// TIA Portal project "Grundkurs Aufgabe 10 NEU" (V15.1)
// Vorlageprojekt für das Buch mit Zielsystem S7-1200

(* hardware
DEVICE "S7-1200-Station_1"  S7-1200 Station
   slot 0: "Baugruppenträger_0"  Rack  V1.0
   slot 1: "SPS"  CPU 1212C AC/DC/Rly  6ES7 212-1BE40-0XB0  V4.2
*)

// ===== PLC "SPS"  CPU 1212C AC/DC/Rly =====

VAR_GLOBAL   // PLC tag table "Eingänge und Ausgänge"
   "Sensor_Bauteil_induktiv" AT %E0.0 : Bool;   // Induktiver Sensor für Werkstofferkennung (Schließer)
   "Sensor_Bauteil_kapazitiv" AT %E0.1 : Bool;   // Kapazitiver Sensor für Werkstofferkennung (Schließer)
   "Endlage_Ausschieber_vorne" AT %E0.2 : Bool;   // Ausschieber hat vorderer Endlage erreicht (Schließer)
   "Endlage_Ausschieber_hinten" AT %E0.3 : Bool;   // Ausschieber hat hintere Endlage erreicht (Schließer)
   "Lichttaster_Auslauf_links" AT %E0.4 : Bool;   // Lichttaster auf Förderband Auslauf links (Schließer)
   "Lichttaster_Auslauf_rechts" AT %E0.5 : Bool;   // Lichttaster auf Förderband Auslauf rechts (Schließer)
   "Motor_Foerderband_Einlauf" AT %A0.0 : Bool;   // Motor Förderband Einlauf vorwärts fahren
   "Motor_Foerderband_Auslauf_links" AT %A0.1 : Bool;   // Motor Förderband Auslauf links vorwärts fahren
   "Motor_Foerderband_Auslauf_rechts" AT %A0.2 : Bool;   // Motor Förderband Auslauf rechts vorwärts fahren
   "Ausschieber_vor" AT %A0.3 : Bool;   // Ausschieber nach vorne fahren (1-Signal = ausfahren / 0-Signal = einfahren)
END_VAR

VAR_GLOBAL   // PLC tag table "Merker"
   "Foerderbaender_Einlauf_Auslauf_vor" AT %M1.0 : Bool;   // Förderbänder Einlauf und Auslauf rechts vorwärts fahren
   "Bauteil_Kunststoff_erkannt" AT %M1.1 : Bool;   // Kunststoffbauteil wurde erkannt
   "Bauteil_Metall_erkannt" AT %M1.2 : Bool;   // Metallbauteil wurde erkannt
   "Bauteil_verschieben" AT %M1.3 : Bool;   // Bauteil auf anderes Förderband verschieben
   "Foerderband_Auslauf_links_vor" AT %M1.4 : Bool;   // Förderband Auslauf links vorwärts fahren
   "Foerderband_Auslauf_rechts_vor" AT %M1.5 : Bool;   // Förderband Auslauf rechts vorwärts fahren
   "Hilfsmerker_FN1" AT %M100.0 : Bool;   // Hilfsmerker für negative Flanke
   "Hilfsmerker_FN2" AT %M100.1 : Bool;   // Hilfsmerker für negative Flanke
   "Hilfsmerker_FN3" AT %M100.2 : Bool;   // Hilfsmerker für negative Flanke
   "Hilfsmerker_FN4" AT %M100.3 : Bool;   // Hilfsmerker für negative Flanke
END_VAR

FUNCTION "Kopplung_FactoryIO_mit_PLCSIM" : Void   // FC9000, SCL
{ S7_Optimized_Access := 'TRUE' }
VERSION : 0.1
   VAR_TEMP
      rdTimeReturn : Int;
      outputTime : DTL;
      SyncVal : Byte;
      forVal : Int;
      forVal_2 : Int;
      Value : Byte;
   END_VAR
   VAR CONSTANT
      CompVal : Byte := 16#34;
      Value_01 : Byte := 16#11;
      Value_01_DW : DWord := 16#A165_D992;
      Value_02_DW : DWord := 16#58BE_4401;
   END_VAR
BEGIN

   #Value:=PEEK(area := 16#82,
        dbNumber := 0,
        byteOffset := 511);
   #Value := #Value + 1;

   POKE(area := 16#82,
        dbNumber := 0,
        byteOffset := 511,
        value := #Value);

   POKE(area:=16#81,
        dbNumber:=0,
        byteOffset:=1016,
        value:=#Value_01_DW);
   POKE(area := 16#81,
        dbNumber := 0,
        byteOffset := 1020,
        value := #Value_02_DW);

   POKE(area := 16#81,
        dbNumber := 0,
        byteOffset := 511,
        value := B#16#00);

   FOR #forVal := 0 TO 120 DO
       FOR #forVal_2:=0 TO 10 DO
           #rdTimeReturn:=RD_SYS_T(#outputTime);
           #rdTimeReturn := WR_SYS_T(#outputTime);
           #rdTimeReturn := RD_SYS_T(#outputTime);
           #rdTimeReturn := WR_SYS_T(#outputTime);
       END_FOR;
       #SyncVal:= PEEK(area := 16#81,
                      dbNumber := 0,
                      byteOffset := 511);
       IF #SyncVal = #CompVal THEN
          GOTO M_1;
       END_IF;
   END_FOR;
   RETURN;

   M_1:
   POKE(area := 16#81,
        dbNumber := 0,
        byteOffset := 511,
        value := B#16#0);
END_FUNCTION

ORGANIZATION_BLOCK "Main"   // OB1, FBD, ProgramCycle
TITLE = "Main Program Sweep (Cycle)"
{ S7_Optimized_Access := 'TRUE' }
VERSION : 0.1
   VAR_INPUT
      Initial_Call : Bool;   // Initial call of this OB
      Remanence : Bool;   // =True, if remanent data are available
   END_VAR
   VAR_TEMP   // added for the SCL form of the ladder/FBD networks
      _w1 : Bool;
   END_VAR
BEGIN

REGION Network 1: Konnektierungsbaustein für PLC-Lab / Bausteinaufruf FC9000 (Für Aufgabe nicht relevant)
   // Im Netzwerk 1 wird der Konnektierungsbaustein für PLC-Lab aufgerufen.
   // Dieser Aufruf darf nicht entfernt werden!
   // Der Baustein FC9000 organisiert den Datentransfer zwischen PLCSIM und FactoryIO.
   // Der Baustein kann als Beispielprojekt von der FactoryIO-Homepage heruntergeladen werden.
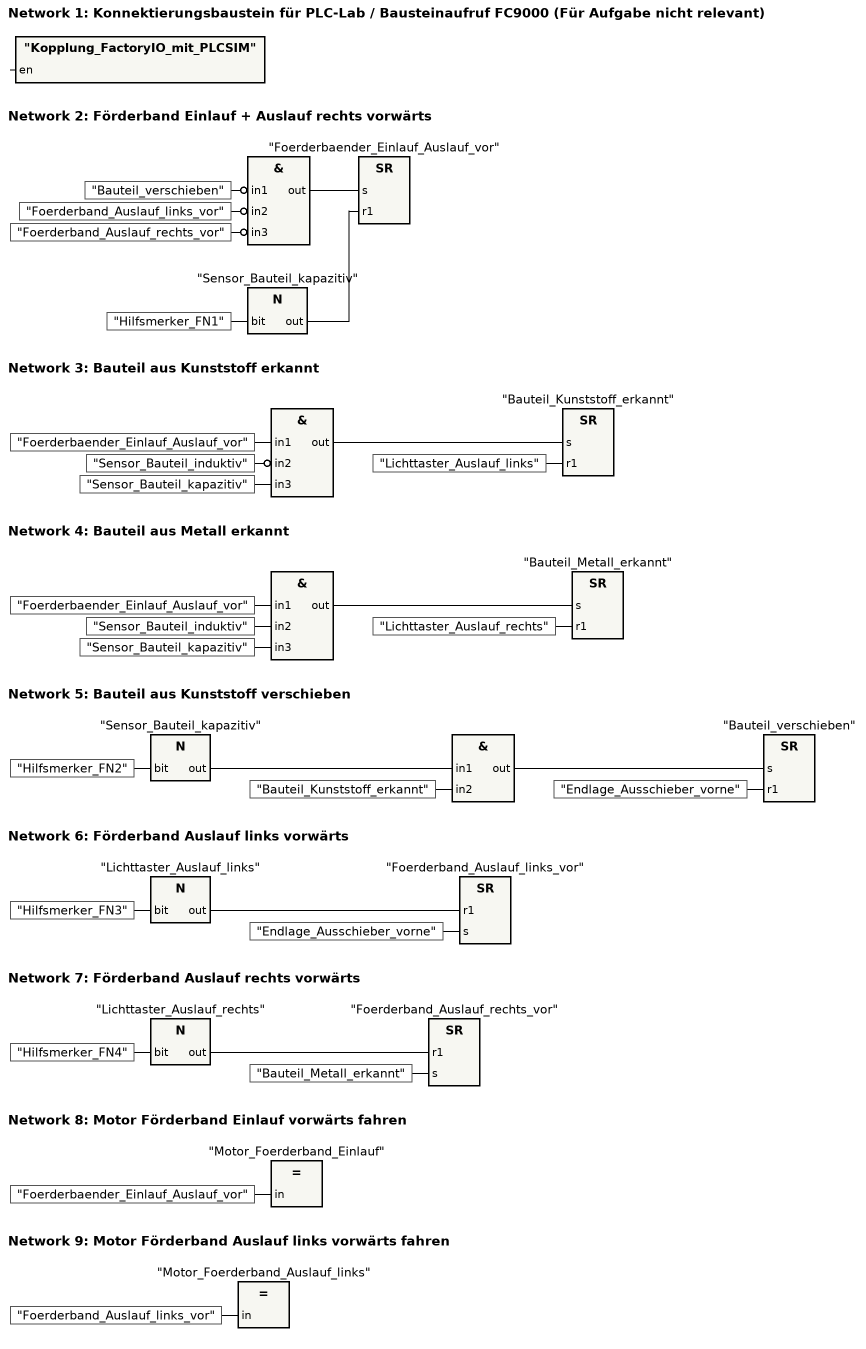
   "Kopplung_FactoryIO_mit_PLCSIM"();
END_REGION

REGION Network 2: Förderband Einlauf + Auslauf rechts vorwärts
   #_w1 := NOT "Sensor_Bauteil_kapazitiv" AND "Hilfsmerker_FN1";   // falling edge of "Sensor_Bauteil_kapazitiv"
   "Hilfsmerker_FN1" := "Sensor_Bauteil_kapazitiv";
   IF NOT "Bauteil_verschieben" AND NOT "Foerderband_Auslauf_links_vor" AND NOT "Foerderband_Auslauf_rechts_vor" THEN
       "Foerderbaender_Einlauf_Auslauf_vor" := TRUE;   // SR flip-flop
   END_IF;
   IF #_w1 THEN "Foerderbaender_Einlauf_Auslauf_vor" := FALSE; END_IF;
END_REGION

REGION Network 3: Bauteil aus Kunststoff erkannt
   IF "Foerderbaender_Einlauf_Auslauf_vor" AND NOT "Sensor_Bauteil_induktiv" AND "Sensor_Bauteil_kapazitiv" THEN
       "Bauteil_Kunststoff_erkannt" := TRUE;   // SR flip-flop
   END_IF;
   IF "Lichttaster_Auslauf_links" THEN "Bauteil_Kunststoff_erkannt" := FALSE; END_IF;
END_REGION

REGION Network 4: Bauteil aus Metall erkannt
   IF "Foerderbaender_Einlauf_Auslauf_vor" AND "Sensor_Bauteil_induktiv" AND "Sensor_Bauteil_kapazitiv" THEN
       "Bauteil_Metall_erkannt" := TRUE;   // SR flip-flop
   END_IF;
   IF "Lichttaster_Auslauf_rechts" THEN "Bauteil_Metall_erkannt" := FALSE; END_IF;
END_REGION

REGION Network 5: Bauteil aus Kunststoff verschieben
   #_w1 := NOT "Sensor_Bauteil_kapazitiv" AND "Hilfsmerker_FN2";   // falling edge of "Sensor_Bauteil_kapazitiv"
   "Hilfsmerker_FN2" := "Sensor_Bauteil_kapazitiv";
   IF #_w1 AND "Bauteil_Kunststoff_erkannt" THEN
       "Bauteil_verschieben" := TRUE;   // SR flip-flop
   END_IF;
   IF "Endlage_Ausschieber_vorne" THEN "Bauteil_verschieben" := FALSE; END_IF;
END_REGION

REGION Network 6: Förderband Auslauf links vorwärts
   #_w1 := NOT "Lichttaster_Auslauf_links" AND "Hilfsmerker_FN3";   // falling edge of "Lichttaster_Auslauf_links"
   "Hilfsmerker_FN3" := "Lichttaster_Auslauf_links";
   IF "Endlage_Ausschieber_vorne" THEN
       "Foerderband_Auslauf_links_vor" := TRUE;   // SR flip-flop
   END_IF;
   IF #_w1 THEN "Foerderband_Auslauf_links_vor" := FALSE; END_IF;
END_REGION

REGION Network 7: Förderband Auslauf rechts vorwärts
   #_w1 := NOT "Lichttaster_Auslauf_rechts" AND "Hilfsmerker_FN4";   // falling edge of "Lichttaster_Auslauf_rechts"
   "Hilfsmerker_FN4" := "Lichttaster_Auslauf_rechts";
   IF "Bauteil_Metall_erkannt" THEN
       "Foerderband_Auslauf_rechts_vor" := TRUE;   // SR flip-flop
   END_IF;
   IF #_w1 THEN "Foerderband_Auslauf_rechts_vor" := FALSE; END_IF;
END_REGION

REGION Network 8: Motor Förderband Einlauf vorwärts fahren
   "Motor_Foerderband_Einlauf" := "Foerderbaender_Einlauf_Auslauf_vor";
END_REGION

REGION Network 9: Motor Förderband Auslauf links vorwärts fahren
   "Motor_Foerderband_Auslauf_links" := "Foerderband_Auslauf_links_vor";
END_REGION

REGION Network 10: Motor Förderband Auslauf rechts vorwärts fahren
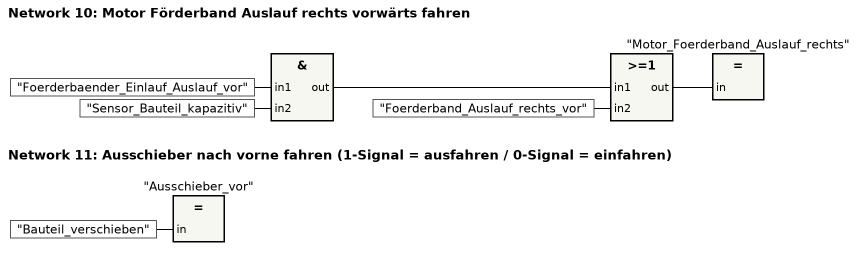
   "Motor_Foerderband_Auslauf_rechts" := ("Foerderbaender_Einlauf_Auslauf_vor" AND "Sensor_Bauteil_kapazitiv") OR "Foerderband_Auslauf_rechts_vor";
END_REGION

REGION Network 11: Ausschieber nach vorne fahren (1-Signal = ausfahren / 0-Signal = einfahren)
   "Ausschieber_vor" := "Bauteil_verschieben";
END_REGION
END_ORGANIZATION_BLOCK